FUNCTION_BLOCK FB_ValueChanged
VAR_INPUT
    Value : INT;
END_VAR
VAR_OUTPUT
    Changed : BOOL;
END_VAR
VAR
    OldValue : INT;
END_VAR

Changed := Value <> OldValue;
OldValue := Value;

END_FUNCTION_BLOCK

(* stored: Version 1.1.0.1, ProductVersion 3.1.4024.3
   POU FB_ValueChanged: Id {fbb70e0f-dba0-4bb1-abc5-028b84aa94a5}, SpecialFunc None *)
